{attribute addProperty BoxType "EJ7342-0000-0019"}
{attribute addProperty Id "ControlAT %Q*Control_197B7E66162"}
{attribute addProperty CRC "1864676036"}
{attribute addProperty SizeInBites "16"}
{attribute addProperty SizeInBytes "2"}
TYPE DCM_Control_Channel_6F24B2C4 :
STRUCT
	{attribute addProperty Name "Control"}
	Control AT %Q* : Control_197B7E66;
END_STRUCT
END_TYPE

(* stored: Version 1.2.0.0, ProductVersion 3.1.4024.9
   DUT DCM_Control_Channel_6F24B2C4: Id {a34ee4cb-600e-4620-8cf9-7bb99aa7ba47} *)
